TYPE E_ResetMode :
(
	AUTO			:=0,	(* Automatic after delay *)
	MANU			:=1	(* Manual *)
);
END_TYPE

(* stored: Version 1.1.0.1, ProductVersion 3.1.4024.9
   DUT E_ResetMode: Id {90f03465-17ea-462b-9183-7dc015bd0b96} *)
